TYPE ST_PowerMonitor_BESS :
STRUCT
	e_ACrotationStatus			: 	eACrotationState;
	ar_Current					:	ARRAY [0..4] OF REAL;
	r_LineVoltage				: 	REAL;
	r_Frequency					: 	REAL;
	r_currentUnbalance			:	REAL;
	//Power
	r_ApparentPower				: 	REAL;
	r_ReactivePower				: 	REAL;
	r_ActivePower				: 	REAL;
	//Energy Consumed
	r_EnergyConsumed			:	REAL;
	
	//Energy Delivered
	r_EnergySupplied			:	REAL;
	
	r_PowerFactor 				:	REAL;
END_STRUCT
END_TYPE

(* stored: Version 1.1.0.1, ProductVersion 3.1.4026.18
   DUT ST_PowerMonitor_BESS: Id {8f4e109a-8fa2-4e4f-b5c9-1b1162dcb21c} *)
